(* PLC project FourceAutomotivePLC, Beckhoff Automation GmbH TwinCAT PLC Control 3.5.13.21 *)
(* stored: creationDateTime 2024-11-06T15:09:09.8286342, modificationDateTime 2024-11-06T15:09:09.8374254 *)

PROGRAM Orderverwerking_magazijn
VAR
	currentState : Task_1 := Task_1.NieuweOrderGaragist;   
	Nieuwe_order: BOOL := TRUE;
	Controleren_voorraad: INT := 0;
	Order_magazijn: BOOL;
	Order_uitgeprint: BOOL;
	Order_verzameld: BOOL; 
	Geannuleerd: BOOL;
	Order_controle: INT :=0;
	Order_voltooid: BOOL;
END_VAR

            CASE currentState OF
    Task_1.NieuweOrderGaragist:
        // Nieuwe bestelling van een garagist
        IF Nieuwe_order = TRUE THEN
            currentState := VoorraadAdministratief;
        END_IF;
		
	Task_1.VoorraadAdministratief:
		// Controleren of de voorraad klopt (Adminastratief)
		IF Controleren_voorraad = 1 THEN
			Order_magazijn := TRUE;
			Order_uitgeprint := TRUE;
			Order_verzameld := TRUE;
			Geannuleerd := FALSE;
			currentState := VerzamelingArtikelen;
		ELSIF Controleren_voorraad = 2 THEN
			Order_magazijn := FALSE;
			Order_uitgeprint := FALSE;
			Order_verzameld := FALSE;
			Geannuleerd := TRUE;
		END_IF
	
		
	Task_1.VerzamelingArtikelen:
	// Controleren of de verzamelde artikelen overeenkomen met de Orderverzamellijst
		IF Order_controle = 1 THEN
			Order_voltooid := TRUE;
			Geannuleerd := FALSE;
		ELSIF Order_controle = 2 THEN
			Order_controle := 0;
			Order_voltooid := FALSE;
			Geannuleerd := FALSE;
		ELSIF Order_controle = 3 THEN
			Order_voltooid := FALSE;
			Geannuleerd := TRUE;			
		END_IF
		
END_CASE;
          
END_PROGRAM
